VAR_GLOBAL
		fbQa:FB_Qa;
		fbIa:FB_Ia;
END_VAR

(* stored: Version 1.1.0.1, ProductVersion 3.1.4020.6
   GVL GVL: Id {1e7ef6ab-0025-4e7c-bbe7-488b25ba0afa} *)
